// TIA Portal V17 export
TagTable "Codex_Popup_Sim_Tags"
  Sim_SelectedCompID : Int  (1 s)   // Sim input: selected component ID, 1=Valve01, 2=Heater01, 3=Fan01
  Sim_ClickPulse : Int  (1 s)   // Sim input: button trigger pulse, 0/1
  Sim_DoubleClickTime_ms : Int  (1 s)   // Sim input: double-click time, default 800 ms
  Sim_Switch1 : Int  (1 s)   // Sim input: Switch[1], 0/1
  Sim_RealValue1 : Real  (1 s)   // Sim input: RealValue[1]
  Sim_Visible : Int  (1 s)   // Sim output: ActivePopup.Visible, 0/1
  Sim_ActiveID : Int  (1 s)   // Sim output: ActivePopup.ActiveID
  Sim_Confirmed : Int  (1 s)   // Sim output: ActivePopup.Confirmed, 0/1
  Sim_ConfirmPulse : Int  (1 s)   // Sim input: ConfirmBtn, 0/1
  Sim_CancelPulse : Int  (1 s)   // Sim input: CancelBtn, 0/1
  Sim_InfoTitle : WString  (1 s)   // Sim output: InfoTitle; editable test text
  Sim_InfoMessage : WString  (1 s)   // Sim output: InfoMessage; editable test text
